Staubli VAL3: colSum.pgx

public program colSum(num& x_nInput[] (dimensions=2), num& x_nResult[])
  local num l_nCols
  local num l_nRows
  local num l_nElement[2]
begin

  l_nRows = size(x_nInput,1)
  l_nCols = size(x_nInput,2)

  resize(x_nResult,1,1)
  x_nResult = 0
  resize(x_nResult,1,l_nCols)

  for l_nElement[0] = 0 to l_nCols-1
    for l_nElement[1] = 0 to l_nRows-1
      x_nResult[l_nElement[0]] = x_nResult[l_nElement[0]] + x_nInput[l_nElement[1],l_nElement[0]]
    endFor
  endFor



end
